TYPE ST_MessageItem :
STRUCT
	/// time stamp
	dtTimeStamp: DT;
	/// priority info, warning, error
	nPriority: BYTE;
	/// message string
	sMessage: T_MaxString;
END_STRUCT
END_TYPE

(* stored: Version 1.1.0.1, ProductVersion 3.1.4024.12
   DUT ST_MessageItem: Id {c276b3e3-ed18-4369-a6ed-db57cf56f410} *)
